{attribute 'linkalways'} 
{attribute 'no_explicit_call' := 'This FB is a CLASS and must be accessed using methods or properties'}
{attribute 'enable_dynamic_creation'}
FUNCTION_BLOCK FINAL AND_BOOL EXTENDS Node
VAR
	in1 : _BOOL(FALSE);
	in2 : _BOOL(FALSE);
	out : _BOOL(FALSE);
END_VAR

METHOD PUBLIC Clone : I_Node
VAR
	pNode : POINTER TO AND_BOOL;
END_VAR
pNode := __NEW(AND_BOOL);
Clone := pNode^;
END_METHOD

METHOD FB_init : BOOL
VAR_INPUT
	bInitRetains : BOOL; // if TRUE, the retain variables are initialized (warm start / cold start)
	bInCopyCode : BOOL;  // if TRUE, the instance afterwards gets moved into the copy code (online change)
END_VAR
AddInput('in1',THIS^.in1);
AddInput('in2',THIS^.in2);
AddOutput('out', THIS^.out);
END_METHOD

METHOD PROTECTED OnExecute
VAR
END_VAR
out.Value := in1.Value AND in2.Value;
END_METHOD

END_FUNCTION_BLOCK

(* stored: Version 1.1.0.1, ProductVersion 3.1.4024.15
   POU AND_BOOL: Id {40ead4d0-b057-4ed2-867e-43ce53033fef}, SpecialFunc None
   Folder Constructor: Id {05a1c20e-1939-4241-bf09-d0e0d3bf2b08}
   Method Clone: Id {d4388e16-073a-4d3d-928d-03b6b57d95fe}
   Method FB_init: Id {629ecbd3-542e-4ebc-ad3e-48f522075313}
   Method OnExecute: Id {50e84d1a-0840-4c4a-a2dc-f502f3010a73} *)
